TYPE ST_BusRelais16F_Cnt :
STRUCT
	dwCntRelais    :ARRAY[1..16] OF DWORD;
END_STRUCT
END_TYPE

(* stored: Version 1.1.0.1, ProductVersion 3.1.4024.12
   DUT ST_BusRelais16F_Cnt: Id {7359cd92-a43a-4e23-800b-501102589fd6} *)
